TYPE SubscriberCell :
STRUCT
	occupied	: BOOL;
	sTopic	   	: STRING;
	sInstance	: STRING;
	subscriber 	: I_SubCallback;
END_STRUCT
END_TYPE

(* stored: Version 1.1.0.1, ProductVersion 3.1.4024.12
   DUT SubscriberCell: Id {dbe08e15-f1a6-4e9a-b884-20bd7fabd328} *)
